// Mitsubishi GX Works2 project: 2023-06-09 #1 생산자동화기능사 16번   PLC: Q03UDV
// 생산자동화기능사

// global labels: Global1
VAR_GLOBAL
  PB1 AT X0 : BOOL;
  PB2 AT X1 : BOOL;
  정지 AT X2 : BOOL;
  공급후진 AT X3 : BOOL;
  공급전진 AT X4 : BOOL;
  가공후진 AT X5 : BOOL;
  가공전진 AT X6 : BOOL;
  송출후진 AT X7 : BOOL;
  송출전진 AT X8 : BOOL;
  배출후진 AT X9 : BOOL;
  배출전진 AT X0A : BOOL;
  매거진 AT X0B : BOOL;
  금속센서 AT X0F : BOOL;
  PB3 AT X0C : BOOL;
  적 AT Y20 : BOOL;
  황 AT Y21 : BOOL;
  녹 AT Y22 : BOOL;
  공급1 AT Y23 : BOOL;
  공급2 AT Y24 : BOOL;
  가공 AT Y25 : BOOL;
  드릴 AT Y26 : BOOL;
  송출 AT Y27 : BOOL;
  배출 AT Y28 : BOOL;
  컨베이어 AT Y29 : BOOL;
END_VAR

PROGRAM 테스트동작
VAR
  PHASE : INT;
END_VAR
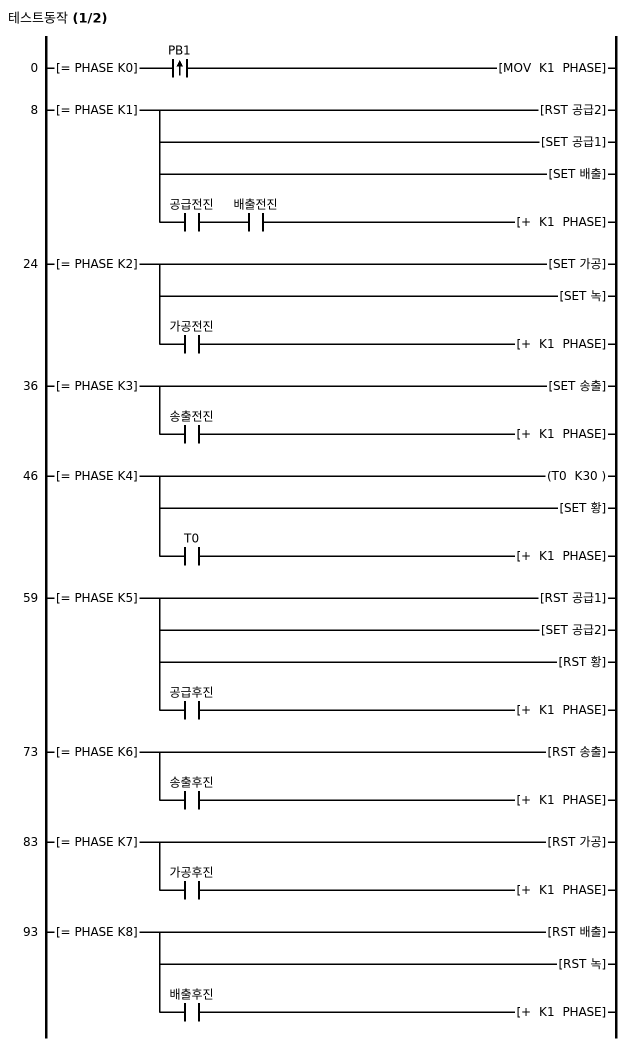
0     LD=     PHASE K0
      ANDP    PB1
      MOV     K1 PHASE
8     LD=     PHASE K1
      RST     공급2
      SET     공급1
      SET     배출
      AND     공급전진
      AND     배출전진
      +       K1 PHASE
24    LD=     PHASE K2
      SET     가공
      SET     녹
      AND     가공전진
      +       K1 PHASE
36    LD=     PHASE K3
      SET     송출
      AND     송출전진
      +       K1 PHASE
46    LD=     PHASE K4
      OUT     T0 K30
      SET     황
      AND     T0
      +       K1 PHASE
59    LD=     PHASE K5
      RST     공급1
      SET     공급2
      RST     황
      AND     공급후진
      +       K1 PHASE
73    LD=     PHASE K6
      RST     송출
      AND     송출후진
      +       K1 PHASE
83    LD=     PHASE K7
      RST     가공
      AND     가공후진
      +       K1 PHASE
93    LD=     PHASE K8
      RST     배출
      RST     녹
      AND     배출후진
      +       K1 PHASE
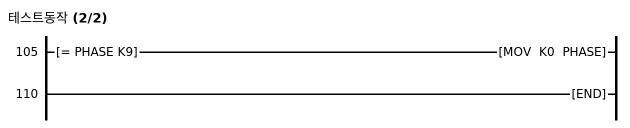
105   LD=     PHASE K9
      MOV     K0 PHASE
110   END
END_PROGRAM

PROGRAM 생산자동화기능사
VAR
  PHASE : INT;
  MODE : INT;
END_VAR
VAR CONSTANT
  단속 : INT;
  연속 : INT := 1;
END_VAR
VAR
  METAL : INT;
END_VAR
VAR CONSTANT
  금속 : INT := 1;
  비금속 : INT := 2;
END_VAR
VAR
  BLINK1 : ARRAY [0..3] OF BOOL;
  STORE : BOOL;
  EMG : INT;
  PHASE1 : INT;
  드릴1 : BOOL;
  컨베이어1 : BOOL;
  녹1 : BOOL;
  황1 : BOOL;
END_VAR
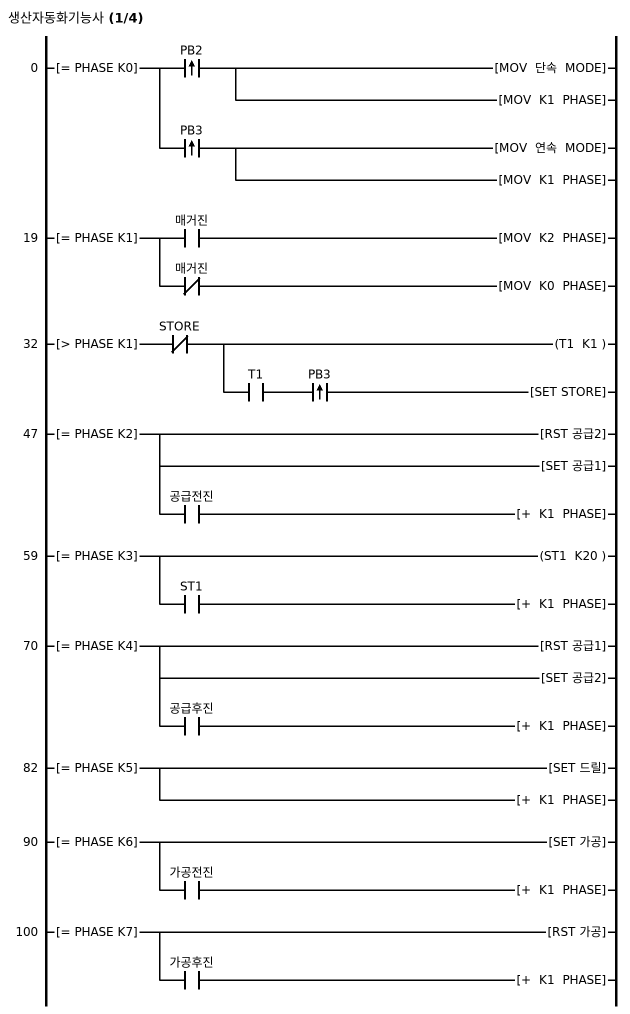
0     LD=     PHASE K0
      MPS
      ANDP    PB2
      MOV     단속 MODE
      MOV     K1 PHASE
      MPP
      ANDP    PB3
      MOV     연속 MODE
      MOV     K1 PHASE
19    LD=     PHASE K1
      MPS
      AND     매거진
      MOV     K2 PHASE
      MPP
      ANI     매거진
      MOV     K0 PHASE
32    LD>     PHASE K1
      ANI     STORE
      OUT     T1 K1
      AND     T1
      ANDP    PB3
      SET     STORE
47    LD=     PHASE K2
      RST     공급2
      SET     공급1
      AND     공급전진
      +       K1 PHASE
59    LD=     PHASE K3
      OUT     ST1 K20
      AND     ST1
      +       K1 PHASE
70    LD=     PHASE K4
      RST     공급1
      SET     공급2
      AND     공급후진
      +       K1 PHASE
82    LD=     PHASE K5
      SET     드릴
      +       K1 PHASE
90    LD=     PHASE K6
      SET     가공
      AND     가공전진
      +       K1 PHASE
100   LD=     PHASE K7
      RST     가공
      AND     가공후진
      +       K1 PHASE
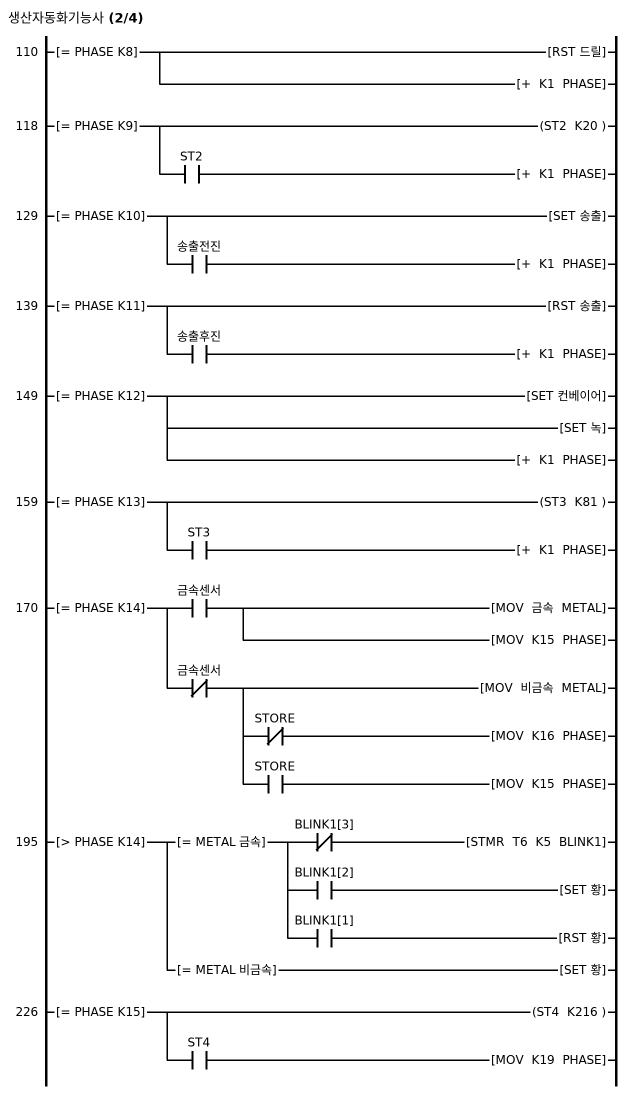
110   LD=     PHASE K8
      RST     드릴
      +       K1 PHASE
118   LD=     PHASE K9
      OUT     ST2 K20
      AND     ST2
      +       K1 PHASE
129   LD=     PHASE K10
      SET     송출
      AND     송출전진
      +       K1 PHASE
139   LD=     PHASE K11
      RST     송출
      AND     송출후진
      +       K1 PHASE
149   LD=     PHASE K12
      SET     컨베이어
      SET     녹
      +       K1 PHASE
159   LD=     PHASE K13
      OUT     ST3 K81
      AND     ST3
      +       K1 PHASE
170   LD=     PHASE K14
      MPS
      AND     금속센서
      MOV     금속 METAL
      MOV     K15 PHASE
      MPP
      ANI     금속센서
      MOV     비금속 METAL
      MPS
      ANI     STORE
      MOV     K16 PHASE
      MPP
      AND     STORE
      MOV     K15 PHASE
195   LD>     PHASE K14
      MPS
      AND=    METAL 금속
      MPS
      ANI     BLINK1[3]
      STMR    T6 K5 BLINK1
      MRD
      AND     BLINK1[2]
      SET     황
      MPP
      AND     BLINK1[1]
      RST     황
      MPP
      AND=    METAL 비금속
      SET     황
226   LD=     PHASE K15
      OUT     ST4 K216
      AND     ST4
      MOV     K19 PHASE
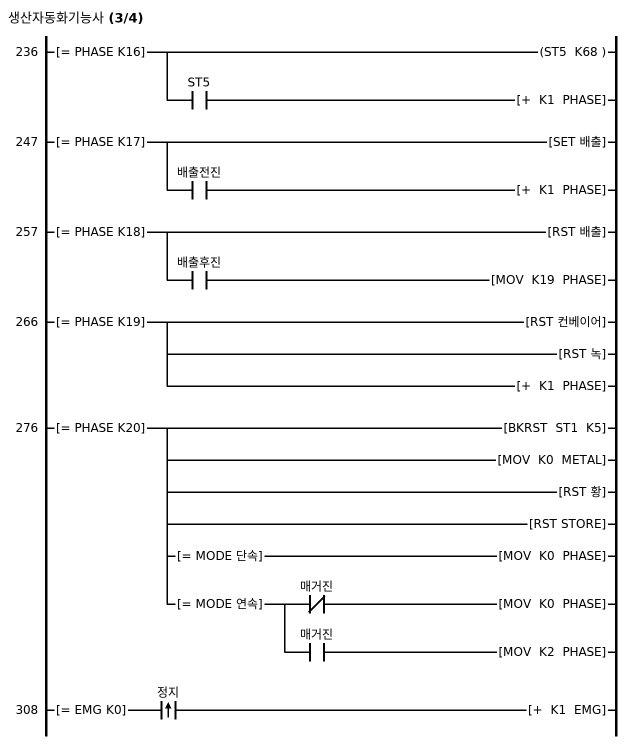
236   LD=     PHASE K16
      OUT     ST5 K68
      AND     ST5
      +       K1 PHASE
247   LD=     PHASE K17
      SET     배출
      AND     배출전진
      +       K1 PHASE
257   LD=     PHASE K18
      RST     배출
      AND     배출후진
      MOV     K19 PHASE
266   LD=     PHASE K19
      RST     컨베이어
      RST     녹
      +       K1 PHASE
276   LD=     PHASE K20
      BKRST   ST1 K5
      MOV     K0 METAL
      RST     황
      RST     STORE
      MPS
      AND=    MODE 단속
      MOV     K0 PHASE
      MPP
      AND=    MODE 연속
      MPS
      ANI     매거진
      MOV     K0 PHASE
      MPP
      AND     매거진
      MOV     K2 PHASE
308   LD=     EMG K0
      ANDP    정지
      +       K1 EMG
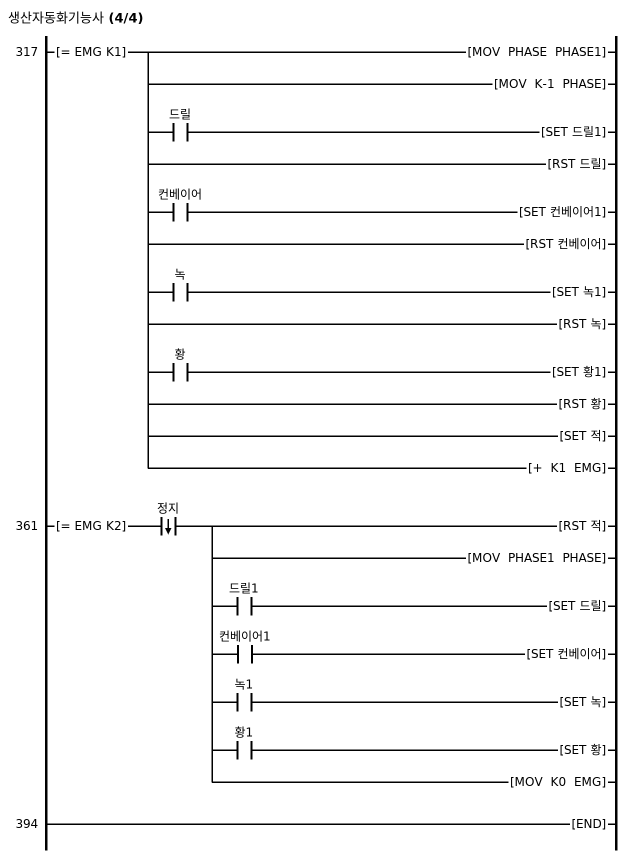
317   LD=     EMG K1
      MOV     PHASE PHASE1
      MOV     K-1 PHASE
      MPS
      AND     드릴
      SET     드릴1
      MPP
      RST     드릴
      MPS
      AND     컨베이어
      SET     컨베이어1
      MPP
      RST     컨베이어
      MPS
      AND     녹
      SET     녹1
      MPP
      RST     녹
      MPS
      AND     황
      SET     황1
      MPP
      RST     황
      SET     적
      +       K1 EMG
361   LD=     EMG K2
      ANDF    정지
      RST     적
      MOV     PHASE1 PHASE
      MPS
      AND     드릴1
      SET     드릴
      MRD
      AND     컨베이어1
      SET     컨베이어
      MRD
      AND     녹1
      SET     녹
      MRD
      AND     황1
      SET     황
      MPP
      MOV     K0 EMG
394   END
END_PROGRAM
